FUNCTION_BLOCK FB_ExitSortingConveyors
VAR_INPUT
	bStop : BOOL;
	bEmgStop : BOOL;
END_VAR
VAR_OUTPUT
END_VAR
VAR
	dummy : BOOL;
	
	CounterLeft : Tc2_Standard.CTU;
	CounterRight : Tc2_Standard.CTU;
	CounterForward : Tc2_Standard.CTU;
END_VAR

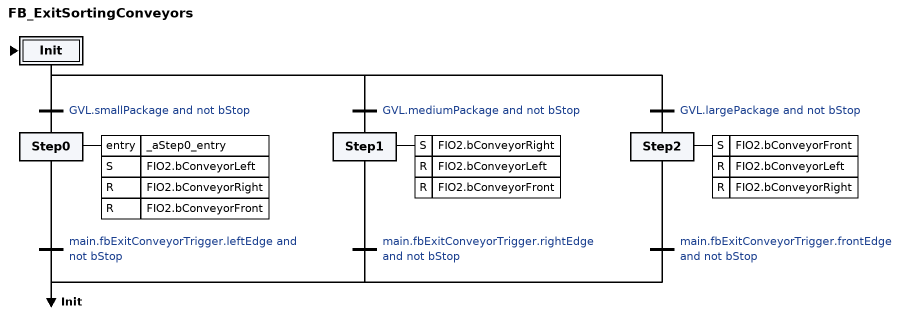
INITIAL_STEP Init:
END_STEP
TRANSITION FROM Init TO Step0
    := GVL.smallPackage and not bStop;
END_TRANSITION
STEP Step0:
    _aStep0_entry(P1);  // entry action
    FIO2.bConveyorLeft(S);
    FIO2.bConveyorRight(R);
    FIO2.bConveyorFront(R);
END_STEP
TRANSITION FROM Step0 TO Init
    := main.fbExitConveyorTrigger.leftEdge and not bStop;
END_TRANSITION
TRANSITION FROM Init TO Step1
    := GVL.mediumPackage and not bStop;
END_TRANSITION
STEP Step1:
    FIO2.bConveyorRight(S);
    FIO2.bConveyorLeft(R);
    FIO2.bConveyorFront(R);
END_STEP
TRANSITION FROM Step1 TO Init
    := main.fbExitConveyorTrigger.rightEdge and not bStop;
END_TRANSITION
TRANSITION FROM Init TO Step2
    := GVL.largePackage and not bStop;
END_TRANSITION
STEP Step2:
    FIO2.bConveyorFront(S);
    FIO2.bConveyorLeft(R);
    FIO2.bConveyorRight(R);
END_STEP
TRANSITION FROM Step2 TO Init
    := main.fbExitConveyorTrigger.frontEdge and not bStop;
END_TRANSITION

END_FUNCTION_BLOCK

(* stored: Version 1.1.0.1, ProductVersion 3.1.4024.13
   POU FB_ExitSortingConveyors: Id {e96b4d14-7028-4e69-b90f-be39a1956bd5}, SpecialFunc None *)
